// Mitsubishi GX Works2 project: MyProject-PLC-new   PLC: FX3U/FX3UC

PROGRAM MAIN
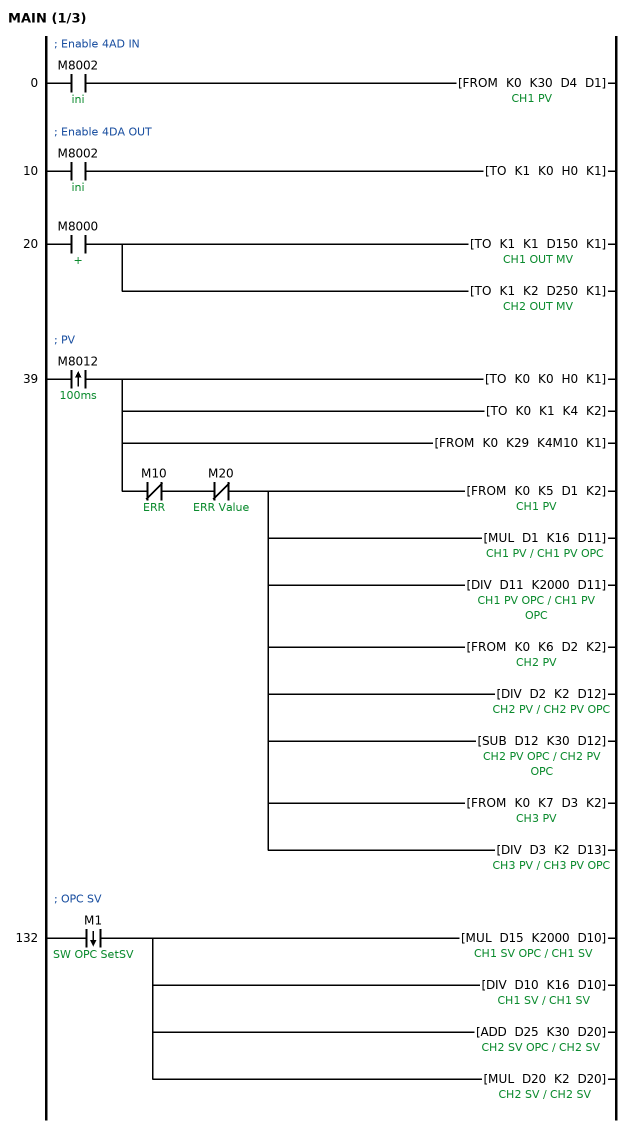
; Enable 4AD IN
0     LD      M8002  ; ini
      FROM    K0 K30 D4 D1  ; CH1 PV
; Enable 4DA OUT
10    LD      M8002  ; ini
      TO      K1 K0 H0 K1
20    LD      M8000  ; +
      TO      K1 K1 D150 K1  ; CH1 OUT MV
      TO      K1 K2 D250 K1  ; CH2 OUT MV
; PV
39    LDP     M8012  ; 100ms
      TO      K0 K0 H0 K1
      TO      K0 K1 K4 K2
      FROM    K0 K29 K4M10 K1  ; ERR
      ANI     M10  ; ERR
      ANI     M20  ; ERR Value
      FROM    K0 K5 D1 K2
      MUL     D1 K16 D11  ; CH1 PV OPC
      DIV     D11 K2000 D11
      FROM    K0 K6 D2 K2  ; CH2 PV
      DIV     D2 K2 D12  ; CH2 PV OPC
      SUB     D12 K30 D12
      FROM    K0 K7 D3 K2  ; CH3 PV
      DIV     D3 K2 D13  ; CH3 PV OPC
; OPC SV
132   LDF     M1  ; SW OPC SetSV
      MUL     D15 K2000 D10  ; CH1 SV OPC / CH1 SV
      DIV     D10 K16 D10
      ADD     D25 K30 D20  ; CH2 SV OPC / CH2 SV
      MUL     D20 K2 D20
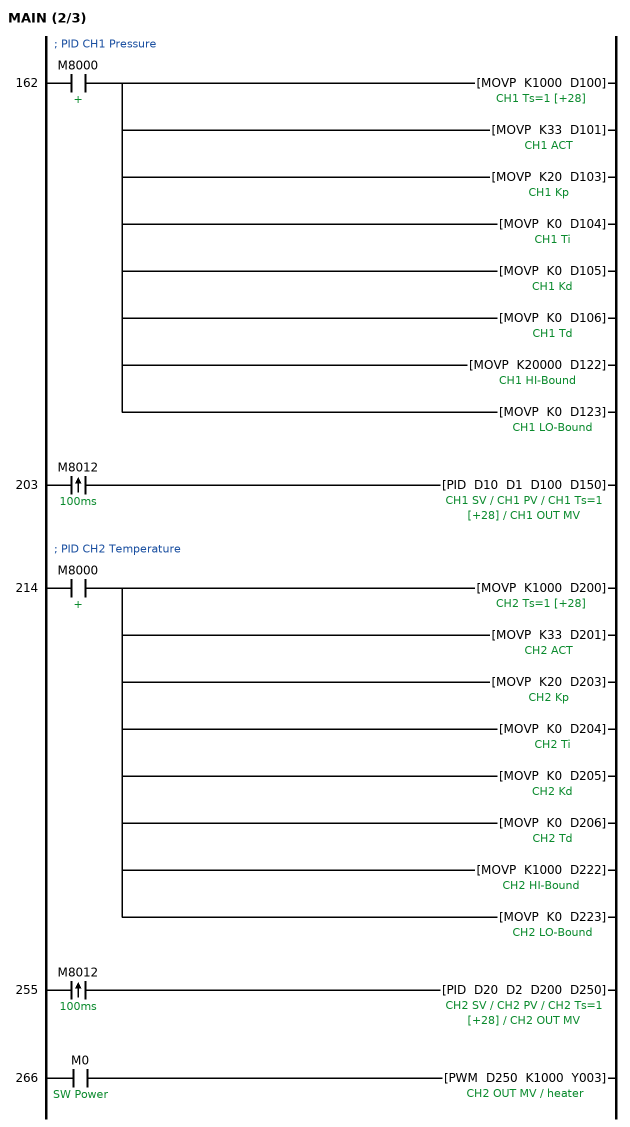
; PID CH1 Pressure
162   LD      M8000  ; +
      MOVP    K1000 D100  ; CH1 Ts=1 [+28]
      MOVP    K33 D101  ; CH1 ACT
      MOVP    K20 D103  ; CH1 Kp
      MOVP    K0 D104  ; CH1 Ti
      MOVP    K0 D105  ; CH1 Kd
      MOVP    K0 D106  ; CH1 Td
      MOVP    K20000 D122  ; CH1 HI-Bound
      MOVP    K0 D123  ; CH1 LO-Bound
203   LDP     M8012  ; 100ms
      PID     D10 D1 D100 D150
; PID CH2 Temperature
214   LD      M8000  ; +
      MOVP    K1000 D200  ; CH2 Ts=1 [+28]
      MOVP    K33 D201  ; CH2 ACT
      MOVP    K20 D203  ; CH2 Kp
      MOVP    K0 D204  ; CH2 Ti
      MOVP    K0 D205  ; CH2 Kd
      MOVP    K0 D206  ; CH2 Td
      MOVP    K1000 D222  ; CH2 HI-Bound
      MOVP    K0 D223  ; CH2 LO-Bound
255   LDP     M8012  ; 100ms
      PID     D20 D2 D200 D250
266   LD      M0  ; SW Power
      PWM     D250 K1000 Y003  ; heater
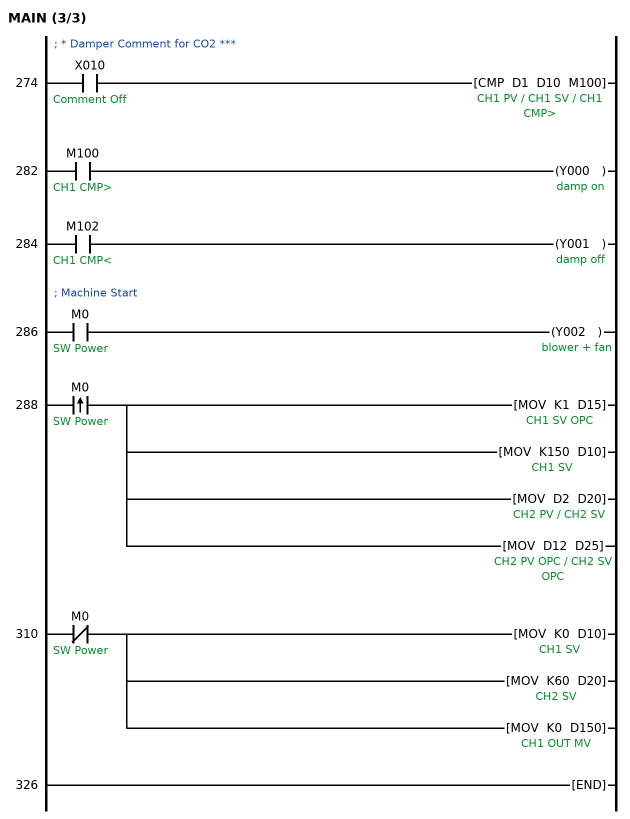
; * Damper Comment for CO2 ***
274   LD      X010  ; Comment Off
      CMP     D1 D10 M100  ; CH1 CMP>
282   LD      M100  ; CH1 CMP>
      OUT     Y000  ; damp on
284   LD      M102  ; CH1 CMP<
      OUT     Y001  ; damp off
; Machine Start
286   LD      M0  ; SW Power
      OUT     Y002  ; blower + fan
288   LDP     M0  ; SW Power
      MOV     K1 D15
      MOV     K150 D10
      MOV     D2 D20
      MOV     D12 D25
310   LDI     M0  ; SW Power
      MOV     K0 D10
      MOV     K60 D20
      MOV     K0 D150
326   END
END_PROGRAM

// device comments not shown above
M101  ; CH1 CMP=
M555  ; comment
